FUNCTION F_LogA4 
VAR_INPUT
	eLogLevel		: E_LogLevel;
	sMessage		: T_MaxString;
	aArg1			: ANY;
	aArg2			: ANY;
	aArg3			: ANY;
	aArg4			: ANY;
END_VAR

F_LogLA4(eLogLevel, Const.sGlobalLogger, sMessage, aArg1, aArg2, aArg3, aArg4);

END_FUNCTION

(* stored: Version 1.1.0.1, ProductVersion 3.1.4024.0
   POU F_LogA4: Id {b475b006-ce64-4702-9a25-2a375136816b}, SpecialFunc None *)
